// TwinCAT 3 PLC project Untitled1
// ProgramVersion: 3.1.4024.0
// libraries:
//   Tc2_Standard, * (Beckhoff Automation GmbH)
//   Tc2_System, * (Beckhoff Automation GmbH)
//   Tc2_Utilities, * (Beckhoff Automation GmbH)
//   Tc3_Module, * (Beckhoff Automation GmbH)
//   TcUnit, * (www.tcunit.org)
// project tree:
//   Common/ StepTimeOutTimer.TcPOU
//   Log/CreateFolder/ CalculateTimeStruct.TcPOU (not stored), FB_CreateFolder.TcPOU, FB_DirectoryControl.TcPOU (not stored), FB_UpdateCurrentSystemTime.TcPOU, F_GetDayOfWeek.TcPOU
//   Log/CreateFolder/DUT/ CreateDirBusy.TcDUT, MethodStatus.TcDUT (not stored), ST_CreateDirBusy.TcDUT (not stored)
//   / PlcTask.TcTTO, ReadMe.TcPOU
//   POUs/ CreateFolder.TcPOU, MAIN.TcPOU
//   TcUnit/ FB_DirectoryContorlTest.TcPOU, POU_Test.TcPOU
// real-time tasks:
//   TASK PlcTask: cycle T#10ms, priority 20, ADS port 350

CONFIGURATION Untitled1
    RESOURCE PLC ON TwinCAT3
        TASK PlcTask(INTERVAL := T#10ms, PRIORITY := 20);
        PROGRAM MAIN WITH PlcTask : MAIN;
    END_RESOURCE
END_CONFIGURATION

// ---- Log/CreateFolder/DUT/CreateDirBusy.TcDUT
TYPE CreateDirBusy :
UNION
	stCreateDirBusy : ST_CreateDirBusy;
	bitCalculator : BYTE;
END_UNION
END_TYPE

// ---- POUs/MAIN.TcPOU
PROGRAM MAIN
VAR
	
END_VAR

CreateFolder();

END_PROGRAM

// ---- POUs/CreateFolder.TcPOU
PROGRAM CreateFolder
VAR
	fbCreateFolder : FB_CreateFolder(sNetID := '', sBasePath := 'C:\createFoldertest\');
	fbUpdateSystemTime : FB_UpdateCurrentSystemTime;
	sPathTest : T_MaxString  := 'C:\test';
	step : INT;
	TimeStruct : TIMESTRUCT;
	bInit: BOOL;
	calTimeStruct : CalculateTimeStruct;
	bTest: BOOL;
END_VAR

fbUpdateSystemTime();
IF bInit THEN
	bInit := FALSE;
	TIMESTRUCT := fbUpdateSystemTime.updatedSystemTime;
END_IF

CASE step OF
	5:
		fbCreateFolder.SetTimeStruct(TIMESTRUCT);
		fbCreateFolder.CreateYearFolder();
		IF fbCreateFolder.isCreatedYearFolder THEN
			step := 8;
		END_IF
	
	6:
		fbCreateFolder.SetTimeStruct(TIMESTRUCT);
		fbCreateFolder.CreateYearMonthDayFolder();
		IF fbCreateFolder.isCreatedYearMonthDayFolder THEN
			step := 8;
		END_IF
	
	7:
		fbCreateFolder.SetTimeStruct(TIMESTRUCT);
		fbCreateFolder.CreateYearMonthFolder();	
		IF fbCreateFolder.isCreatedYearMonthFolder THEN
			step := 8;
		END_IF
	
	8: (* Increase Month or Year or Day for Test *)
		TIMESTRUCT.wYear := TIMESTRUCT.wYear + 1;
		calTimeStruct(TimeStruct := TimeStruct);
		step := 5;	
END_CASE

END_PROGRAM

// ---- Log/CreateFolder/FB_CreateFolder.TcPOU
(* Call SetTimeStruct method before create any folder *)

FUNCTION_BLOCK FB_CreateFolder
VAR_INPUT
	sNetID : T_AmsNetId :='';
	sBasePath : T_MaxString := 'C:\logs\'; // Last of Path needs to have '\'
END_VAR
VAR_OUTPUT
	isCreatedYearFolder : BOOL;
	isCreatedYearMonthDayFolder : BOOL;
	isCreatedYearMonthFolder : BOOL;
END_VAR
VAR
	updatedSystemTime : TIMESTRUCT; 
	fbDirectoryControl : FB_DirectoryControl;
	CreateDirBusy : CreateDirBusy;
END_VAR

METHOD CreateYearFolder
VAR_INPUT
END_VAR
VAR
	sPath : T_MaxString;
END_VAR

VAR_INST
	sFileName : STRING(20);
	step : INT := 10;
	TimeOutTimer : StepTimeOutTimer;
END_VAR
TimeOutTimer(step := step);
IF TimeOutTimer.hasTimeOut THEN
	StepReset(step := step);
END_IF

IF NOT(CreateDirBusy.bitCalculator = 0 OR CreateDirBusy.stCreateDirBusy.isYearBusy = TRUE) THEN
	RETURN;
END_IF

CASE step OF
	0:
		CreateDirBusy.stCreateDirBusy.isYearBusy := FALSE;
		isCreatedYearFolder := FALSE;
		step := 10;
	10:
		CreateDirBusy.stCreateDirBusy.isYearBusy := TRUE;
		
		sFileName := CONCAT(WORD_TO_STRING(updatedSystemTime.wYear), 'Y');
		sPath := CONCAT(sBasePath, sFileName);
		
		fbDirectoryControl.CreateDirectory(sPath := sPath);
		IF NOT fbDirectoryCOntrol.CreateDirectoryStatus.Busy THEN
			step := 20;
		END_IF
	20:
		
		fbDirectoryControl.CheckDirectory(sSearchDirectoryPath := sBasePath, sCreatedFolderName := sFileName);
		IF NOT fbDirectoryControl.CheckDirectoryStatus.Busy THEN
			step := 30;
		END_IF
		
	30:
		IF fbDirectoryControl.hasDirecotryChecked THEN
			step := 0;
			isCreatedYearFolder := TRUE;
		ELSE
			step := 10;
		END_IF
END_CASE
END_METHOD

METHOD CreateYearMonthDayFolder

VAR
	sPath : T_MaxString;
END_VAR
VAR_INST
	step : INT;
	sFileName : STRING(20);
	sDayBasePath : T_MaxString;
	TimeOutTimer : StepTimeOutTimer;
END_VAR
TimeOutTimer(step := step);
IF TimeOutTimer.hasTimeOut THEN
	StepReset(step := step);
END_IF

CreateYearMonthFolder();

IF NOT(CreateDirBusy.bitCalculator = 0 OR CreateDirBusy.stCreateDirBusy.isDayBusy = TRUE) THEN
	RETURN;
END_IF

CASE step OF
	0:
		CreateDirBusy.stCreateDirBusy.isDayBusy := FALSE;
		isCreatedYearMonthDayFolder := FALSE;
		step := 100;
	 
	100:
		CreateDirBusy.stCreateDirBusy.isDayBusy := TRUE;
		
		sFileName := CONCAT(WORD_TO_STRING(updatedSystemTime.wDay), 'th');
		sDayBasePath := CONCAT(sBasePath, WORD_TO_STRING(updatedSystemTime.wYear));
		sDayBasePath := CONCAT(sDayBasePath, 'Y' );
		sDayBasePath := CONCAT(sDayBasePath, '\' );
		sDayBasePath := CONCAT(sDayBasePath,F_GetDayOfWeek(updatedSystemTime.wMonth));
		sDayBasePath := CONCAT(sDayBasePath,'\' );
		sPath := CONCAT(sDayBasePath,sFileName);
		
		
		fbDirectoryControl.CreateDirectory(sPath := sPath);
		IF NOT fbDirectoryCOntrol.CreateDirectoryStatus.Busy THEN
			step := 200;
		END_IF
	200:
		fbDirectoryControl.CheckDirectory(sSearchDirectoryPath := sDayBasePath, sCreatedFolderName := sFileName);
		IF NOT fbDirectoryControl.CheckDirectoryStatus.Busy THEN
			step := 300;
		END_IF
		
	300:
		IF fbDirectoryControl.hasDirecotryChecked THEN
			step := 0;
			isCreatedYearMonthDayFolder := TRUE; 
		ELSE
			step := 100;
		END_IF
END_CASE
END_METHOD

METHOD CreateYearMonthFolder
VAR_INPUT
END_VAR

VAR
	sPath : T_MaxString;
END_VAR

VAR_INST
	step : INT;
	sFileName : STRING(20);
	sMonthBasePath : T_MaxString;
	TimeOutTimer : StepTimeOutTimer;
END_VAR
TimeOutTimer(step := step);
IF TimeOutTimer.hasTimeOut THEN
	StepReset(step := step);
END_IF

CreateYearFolder();


IF NOT(CreateDirBusy.bitCalculator = 0 OR CreateDirBusy.stCreateDirBusy.isMonthBusy = TRUE) THEN
	RETURN;
END_IF


CASE step OF
	0:
		CreateDirBusy.stCreateDirBusy.isMonthBusy := FALSE;
		isCreatedYearMonthFolder := FALSE;
		step := 100;
	 
	100:
		CreateDirBusy.stCreateDirBusy.isMonthBusy := TRUE;
		
		sFileName := F_GetDayOfWeek(THIS^.updatedSystemTime.wMonth);
		sMonthBasePath := CONCAT(sBasePath, WORD_TO_STRING(updatedSystemTime.wYear));
		sMonthBasePath := CONCAT(sMonthBasePath, 'Y');
		sMonthBasePath := CONCAT(sMonthBasePath,'\' );
		sPath := CONCAT(sMonthBasePath,sFileName);
		
		
		fbDirectoryControl.CreateDirectory(sPath := sPath);
		IF NOT fbDirectoryCOntrol.CreateDirectoryStatus.Busy THEN
			step := 200;
		END_IF
	200:
		fbDirectoryControl.CheckDirectory(sSearchDirectoryPath := sMonthBasePath, sCreatedFolderName := sFileName);
		IF NOT fbDirectoryControl.CheckDirectoryStatus.Busy THEN
			step := 300;
		END_IF
		
	300:
		IF fbDirectoryControl.hasDirecotryChecked THEN
			step := 0;
			isCreatedYearMonthFolder := TRUE;
		ELSE
			step := 100;
		END_IF
END_CASE
END_METHOD

METHOD FB_init : BOOL
VAR_INPUT
	bInitRetains : BOOL; // if TRUE, the retain variables are initialized (warm start / cold start)
	bInCopyCode : BOOL;  // if TRUE, the instance afterwards gets moved into the copy code (online change)
	sNetID : T_AmsNetId :='';
	sBasePath : T_MaxString := 'C:\logs\'; // Last of Path needs to have '\'
	
END_VAR
THIS^.sNetID := sNetId;
THIS^.sBasePath := sBasePath;
END_METHOD

METHOD SetTimeStruct
VAR_INPUT
	SystemTime : TIMESTRUCT;
END_VAR
(* If this is creating folder time shouldn't be changed *)
IF NOT (THIS^.CreateDirBusy.bitCalculator = 0) THEN
	RETURN;
END_IF

THIS^.updatedSystemTime := SystemTime;
END_METHOD

METHOD StepReset
VAR_INPUT
	Step : REFERENCE TO INT;
END_VAR
step := 0;
This^.CreateDirBusy.bitCalculator := 0;
END_METHOD

END_FUNCTION_BLOCK

// ---- Common/StepTimeOutTimer.TcPOU
FUNCTION_BLOCK StepTimeOutTimer
VAR_IN_OUT
	step : INT;
END_VAR
VAR_INPUT
	TimeOut : TIME := T#30S;
END_VAR
VAR_OUTPUT
	hasTimeOut : BOOL;
END_VAR
VAR
	Timer : TON;
	oldStep : INT;
END_VAR

Timer(IN := oldStep = step, PT := TimeOut);
IF Timer.Q THEN
	hasTimeOut := TRUE;
ELSE
	hasTimeOut := FALSE;
END_IF
oldStep := step;

END_FUNCTION_BLOCK

// ---- Log/CreateFolder/F_GetDayOfWeek.TcPOU
FUNCTION F_GetDayOfWeek : STRING(4)
VAR_INPUT
	wMonth : WORD;
END_VAR

CASE wMonth OF
	1:
		F_GetDayOfWeek := 'Jan';
	2:  
		F_GetDayOfWeek := 'Feb';
	3:  
		F_GetDayOfWeek := 'Mar';
	4:  
		F_GetDayOfWeek := 'Apr';
	5:  
		F_GetDayOfWeek := 'May';
	6:  
		F_GetDayOfWeek := 'Jun';
	7:  
		F_GetDayOfWeek := 'Jul';
	8:  
		F_GetDayOfWeek := 'Aug';
	9:  
		F_GetDayOfWeek := 'Sep';
	10: 
		F_GetDayOfWeek := 'Oct';
	11: 
		F_GetDayOfWeek := 'Nov';
	12: 
		F_GetDayOfWeek := 'Dec';
END_CASE

END_FUNCTION

// ---- Log/CreateFolder/FB_UpdateCurrentSystemTime.TcPOU
FUNCTION_BLOCK FB_UpdateCurrentSystemTime
VAR_INPUT
	UpdateDelay: TIME := T#0S;
END_VAR
VAR_OUTPUT
	updatedSystemTime		: TIMESTRUCT;
	UpdatedCount 			: UINT;
END_VAR
VAR
	step 					: INT;
	UpdateTimer			 	: TON;
	GetTime					: NT_GetTime;
END_VAR

CASE step OF
	0:
		GetTime(
		NETID:= , 
		START:= FALSE, 
		TMOUT:= , 
		BUSY=> , 
		ERR=> , 
		ERRID=> , 
		TIMESTR=>updatedSystemTime);
		UpdateTimer(In:=TRUE, PT := UpdateDelay);
		IF UpdateTimer.Q THEN
			step := 10;
			UpdateTimer(In:=FALSE, PT := UpdateDelay);
		END_IF
		
	10:
		GetTime(
		NETID:= , 
		START:= TRUE, 
		TMOUT:= , 
		BUSY=> , 
		ERR=> , 
		ERRID=> , 
		TIMESTR=>updatedSystemTime);
		
		IF NOT GetTime.BUSY THEN
			IF GetTime.ERR THEN
				step := 99;
			ELSE
				step := 20;
			END_IF
		END_IF
	20:
		IF UpdatedCount >= 65500 THEN
			UpdatedCount := 0;
		END_IF
		UpdatedCount := UpdatedCount + 1;
		step := 0;
	99:
		step := 0;
END_CASE

END_FUNCTION_BLOCK

// ---- ReadMe.TcPOU
PROGRAM ReadMe

(*

Function Block
 - InOutput, InPut, Output are intended to use from other program
 - Properties are intended for Encapsulation
































*)

END_PROGRAM

// ---- TcUnit/FB_DirectoryContorlTest.TcPOU
FUNCTION_BLOCK FB_DirectoryContorlTest EXTENDS TcUnit.FB_TestSuite

CreateDictionaryTest();

METHOD CreateDictionaryTest
VAR_INPUT
END_VAR

VAR_INST
	Timer : TON := (PT := T#50S);
	fbDirectoryControl : FB_DirectoryControl;
	bDone : REFERENCE TO BOOL;
END_VAR
IF TEST_ORDERED('CreateDiectionaryTest') THEN
	Timer(In:=TRUE);
	
	
	IF Timer.Q THEN
		
		AssertEquals(Expected := bDone
					,Actual := bDone
					,Message := 'CreateDirectoryFail' );
	
		TEST_FINISHED();
	END_IF
END_IF
END_METHOD

END_FUNCTION_BLOCK

// ---- TcUnit/POU_Test.TcPOU
PROGRAM POU_Test
VAR
	fbDirectoryContorlTest : FB_DirectoryContorlTest;
END_VAR

//TcUnit.RUN();

END_PROGRAM
